// TIA Portal V21 export
// export: Created 2026-05-11T00:00:00.0000000Z, ExportSetting None, DisplayName Totally Integrated Automation Portal, DisplayVersion V21, DisplayName STEP 7 Professional, DisplayVersion V21
FUNCTION "MCPVerify_FC_LAD_v2" : Void   // FC902, LAD
TITLE = MCP LAD 原生指令验证 v2
{ S7_Optimized_Access := 'TRUE' }
// MCP 验证 v2: Eq/Ne/Le/Ge/Sub/Mul/Div/Mod/Convert + 取反触点
// stored: AutoNumber false, SetENOAutomatically false
   VAR_INPUT
      "A" : Bool;
      "B" : Bool;
      V1 : Int;
      V2 : Int;
      R1 : Real;
   END_VAR
   VAR_OUTPUT
      O_EQ : Bool;
      O_NE : Bool;
      O_LE : Bool;
      O_GE : Bool;
      DIFF : Int;
      PROD : Int;
      QUOT : Int;
      REM : Int;
      REAL_OUT : Real;
      O_NEG : Bool;
   END_VAR
BEGIN

REGION Network 1: N1-Eq
   // Eq: V1 == V2 -> O_EQ
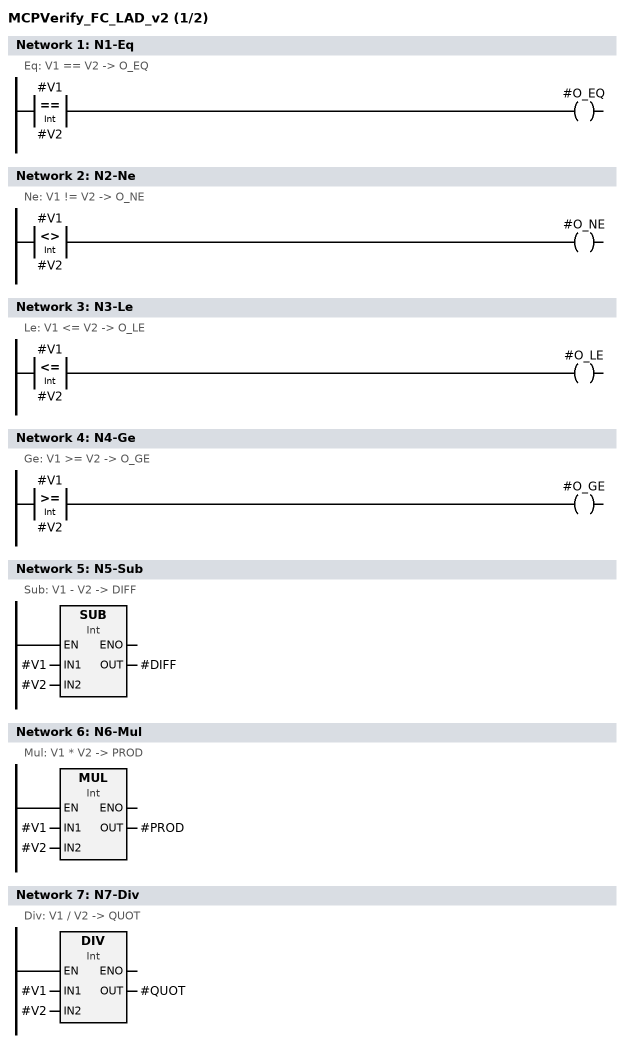
   RUNG wire#powerrail
      { S7_Templates := "SrcType := Int" } EQ_Contact(in1 := #V1, in2 := #V2)
      Coil( #O_EQ )
   END_RUNG
   // the same network as SCL:
   #O_EQ := #V1 = #V2;
END_REGION

REGION Network 2: N2-Ne
   // Ne: V1 != V2 -> O_NE
   RUNG wire#powerrail
      { S7_Templates := "SrcType := Int" } NE_Contact(in1 := #V1, in2 := #V2)
      Coil( #O_NE )
   END_RUNG
   // the same network as SCL:
   #O_NE := #V1 <> #V2;
END_REGION

REGION Network 3: N3-Le
   // Le: V1 <= V2 -> O_LE
   RUNG wire#powerrail
      { S7_Templates := "SrcType := Int" } LE_Contact(in1 := #V1, in2 := #V2)
      Coil( #O_LE )
   END_RUNG
   // the same network as SCL:
   #O_LE := #V1 <= #V2;
END_REGION

REGION Network 4: N4-Ge
   // Ge: V1 >= V2 -> O_GE
   RUNG wire#powerrail
      { S7_Templates := "SrcType := Int" } GE_Contact(in1 := #V1, in2 := #V2)
      Coil( #O_GE )
   END_RUNG
   // the same network as SCL:
   #O_GE := #V1 >= #V2;
END_REGION

REGION Network 5: N5-Sub
   // Sub: V1 - V2 -> DIFF
   RUNG wire#powerrail
      { S7_Templates := "SrcType := Int" } Sub(in1 := #V1, in2 := #V2, out => #DIFF)
   END_RUNG
   // the same network as SCL:
   #DIFF := #V1 - #V2;
END_REGION

REGION Network 6: N6-Mul
   // Mul: V1 * V2 -> PROD
   RUNG wire#powerrail
      { S7_Templates := "SrcType := Int" } Mul(in1 := #V1, in2 := #V2, out => #PROD)
   END_RUNG
   // the same network as SCL:
   #PROD := #V1 * #V2;
END_REGION

REGION Network 7: N7-Div
   // Div: V1 / V2 -> QUOT
   RUNG wire#powerrail
      { S7_Templates := "SrcType := Int" } Div(in1 := #V1, in2 := #V2, out => #QUOT)
   END_RUNG
   // the same network as SCL:
   #QUOT := #V1 / #V2;
END_REGION

REGION Network 8: N8-Mod
   // Mod: V1 mod V2 -> REM
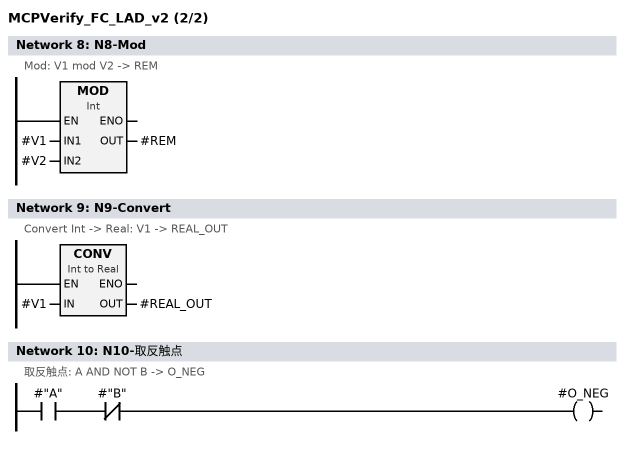
   RUNG wire#powerrail
      { S7_Templates := "SrcType := Int" } Mod(in1 := #V1, in2 := #V2, out => #REM)
   END_RUNG
   // the same network as SCL:
   #REM := #V1 MOD #V2;
END_REGION

REGION Network 9: N9-Convert
   // Convert Int -> Real: V1 -> REAL_OUT
   RUNG wire#powerrail
      { S7_Templates := "[SrcType := Int, DestType := Real]" } Convert(in := #V1, out => #REAL_OUT)
   END_RUNG
   // the same network as SCL:
   #REAL_OUT := INT_TO_REAL(#V1);
END_REGION

REGION Network 10: N10-取反触点
   // 取反触点: A AND NOT B -> O_NEG
   RUNG wire#powerrail
      Contact( #"A" )
      I_Contact( #"B" )
      Coil( #O_NEG )
   END_RUNG
   // the same network as SCL:
   #O_NEG := #"A" AND NOT #"B";
END_REGION
END_FUNCTION
